Fanuc KAREL source: kt00737.KL

-- PROVISIONAL review KL for V940-1; original PC SHA256 0c4e4b9c4a1d34f46683cd9e6ca1003237a53d4df7152fe121cdc75425ad23b8
-- Incomplete behavior may be omitted. Consult companion uncertainty JSON. Do not deploy.
PROGRAM KT00737
%NOLOCKGROUP
BEGIN
  -- V9_ZERO_TABLE_METADATA_HINT layout=0001; no indexed target words; source/name/runtime held
  -- UNRESOLVED_PC offsets 5-18; opcodes 22,1D,23
  -- UNRESOLVED_PC offsets 23-27; opcodes 7F
END KT00737
